PROGRAM MAIN
VAR
	bFirstCycleExecuted : BOOL := FALSE;
	Unit : UNIT_Blikkenvullijn;
//	Devices : FB_Devices;
	
	Start		: BOOL;
	Stop		: BOOL;
	Reset		: BOOL;
	Abort		: BOOL;
	Clear		: BOOL;
	UnSuspend	: BOOL;
	Suspend		: BOOL;
	UnHold		: BOOL;
	Hold		: BOOL;
	Auto		: BOOL;
	Manueel		: BOOL;
END_VAR

(*
$$$$$$$$\                                                                   $$\       $$$$$$$$\                     $$\                                         $$\                     
$$  _____|                                                                  $$ |      $$  _____|                    \__|                                        \__|                    
$$ |   $$$$$$\   $$$$$$\  $$$$$$$\  $$\  $$\  $$\  $$$$$$\   $$$$$$\   $$$$$$$ |      $$ |      $$$$$$$\   $$$$$$\  $$\ $$$$$$$\   $$$$$$\   $$$$$$\   $$$$$$\  $$\ $$$$$$$\   $$$$$$\  
$$$$$\ \____$$\ $$  __$$\ $$  __$$\ $$ | $$ | $$ |$$  __$$\ $$  __$$\ $$  __$$ |      $$$$$\    $$  __$$\ $$  __$$\ $$ |$$  __$$\ $$  __$$\ $$  __$$\ $$  __$$\ $$ |$$  __$$\ $$  __$$\ 
$$  __|$$$$$$$ |$$ |  \__|$$ |  $$ |$$ | $$ | $$ |$$ /  $$ |$$ /  $$ |$$ /  $$ |      $$  __|   $$ |  $$ |$$ /  $$ |$$ |$$ |  $$ |$$$$$$$$ |$$$$$$$$ |$$ |  \__|$$ |$$ |  $$ |$$ /  $$ |
$$ |  $$  __$$ |$$ |      $$ |  $$ |$$ | $$ | $$ |$$ |  $$ |$$ |  $$ |$$ |  $$ |      $$ |      $$ |  $$ |$$ |  $$ |$$ |$$ |  $$ |$$   ____|$$   ____|$$ |      $$ |$$ |  $$ |$$ |  $$ |
$$ |  \$$$$$$$ |$$ |      $$ |  $$ |\$$$$$\$$$$  |\$$$$$$  |\$$$$$$  |\$$$$$$$ |      $$$$$$$$\ $$ |  $$ |\$$$$$$$ |$$ |$$ |  $$ |\$$$$$$$\ \$$$$$$$\ $$ |      $$ |$$ |  $$ |\$$$$$$$ |
\__|   \_______|\__|      \__|  \__| \_____\____/  \______/  \______/  \_______|      \________|\__|  \__| \____$$ |\__|\__|  \__| \_______| \_______|\__|      \__|\__|  \__| \____$$ |
                                                                                                          $$\   $$ |                                                          $$\   $$ |
                                                                                                          \$$$$$$  |                                                          \$$$$$$  |
                                                                                                           \______/                                                            \______/ 
*)

//*****************************UNIT*****************************//
Unit();

//******************************CM******************************//
//Devices();


IF NOT bFirstCycleExecuted THEN
	//Unit
	Unit.FB_init(0,0);
	unit.Auto();	
	bFirstCycleExecuted := TRUE;
END_IF




    // Implement automatic mode logic
IF Start THEN
	unit.start();
	Start := FALSE;
END_IF
    
IF Stop THEN
	unit.stop();
	Stop := FALSE;
END_IF

IF Reset THEN
	Unit.reset();
	Reset := FALSE;
END_IF

IF Abort THEN
	unit.abort();
	Abort := FALSE;
END_IF

IF Clear THEN
	unit.clear();
	Clear := FALSE;
END_IF

IF UnSuspend THEN
	unit.unsuspend();
	UnSuspend := FALSE;
END_IF

IF Suspend THEN
	unit.suspend();
	Suspend := FALSE;
END_IF

IF UnHold THEN
	unit.unhold();
	UnHold := FALSE;
END_IF

IF Hold THEN
	unit.hold();
	Hold := FALSE;
END_IF

IF Auto THEN
	unit.Auto();
	Auto := FALSE;
END_IF

IF Manueel THEN
	unit.Manueel();
	Manueel := FALSE;
END_IF

END_PROGRAM

(* stored: Version 1.1.0.1, ProductVersion 3.1.4024.12
   POU MAIN: Id {8118f260-c6ec-41e8-9a07-ee81d80bcf5e}, SpecialFunc None *)
